PROGRAM prgGrid
VAR
	

	lrPowerGrid		: LREAL;						//{#lynus.ag#()}
	rSizeGridConn		: REAL;							//{#lynus.ag#()}
	lrCounterGridProd			: LREAL;								//{#lynus.ag#()}
	lrCounterGridCons			: LREAL;								//{#lynus.ag#()}

END_VAR

prgGrid.lrPowerGrid				:=	prg_ADS.struct_received.lrPowerGrid			;
prgGrid.rSizeGridConn			:=	prg_ADS.struct_received.rSizeGridConn			;
lrCounterGridProd				:= 	prg_ADS.struct_received.lrCounterGridProd ;
lrCounterGridCons				:= 	prg_ADS.struct_received.lrCounterGridCons	;

END_PROGRAM

(* stored: Version 1.1.0.1, ProductVersion 3.1.4024.12
   POU prgGrid: Id {a8b7bea9-4b66-4291-bbc0-9cb0942a8c9d}, SpecialFunc None *)
